(* CODESYS project Johnson,Joachim,Uppgift16.project

Project tree, tasks and I/O mapping:
  Device : CODESYS Control Win V3, 3S - Smart Software Solutions GmbH, order no. 305021, version 3.5.10.40
    application Application
      libraries: Standard, * (System)
      task MainTask (cyclic, interval t#20ms, priority 1) calls PLC_PRG
      program PLC_PRG [SFC]: MoveConv1to2, MoveCon2to3
      global variables GVL
      Symbols
*)

// Device/Application/GVL
{attribute 'qualified_only'}
VAR_GLOBAL
	// signals
	iSUB01_B1: BOOL; // Signals för conveyor 1. ontop
	iSUB02_B1: BOOL; // Signals för conveyor 2. ontop
	iSUB03_B1: BOOL; // Signals för conveyor 3. ontop
	
	// conveyor signal ontop conveyro.
	oSUB01_K1: BOOL; // MOTOR FÖR converoyr 1
	oSUB02_K1: BOOL; // MOTOR FÖR converoyr 2
	oSUB03_K1: BOOL; // MOTOR FÖR converoyr 3
END_VAR

// Device/Application/PLC_PRG
PROGRAM PLC_PRG
VAR
END_VAR
VAR // added by the converter: edge detectors and wires of the graphical bodies
    _w1, _w3 : BOOL;
    _w2 : ANY;
END_VAR

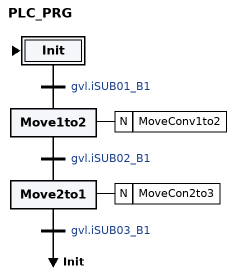
INITIAL_STEP Init:
END_STEP
TRANSITION FROM Init TO Move1to2
    := gvl.iSUB01_B1;
END_TRANSITION
STEP Move1to2:
    MoveConv1to2(N);
END_STEP
TRANSITION FROM Move1to2 TO Move2to1
    := gvl.iSUB02_B1;
END_TRANSITION
STEP Move2to1:
    MoveCon2to3(N);
END_STEP
TRANSITION FROM Move2to1 TO Init
    := gvl.iSUB03_B1;
END_TRANSITION

ACTION MoveConv1to2:
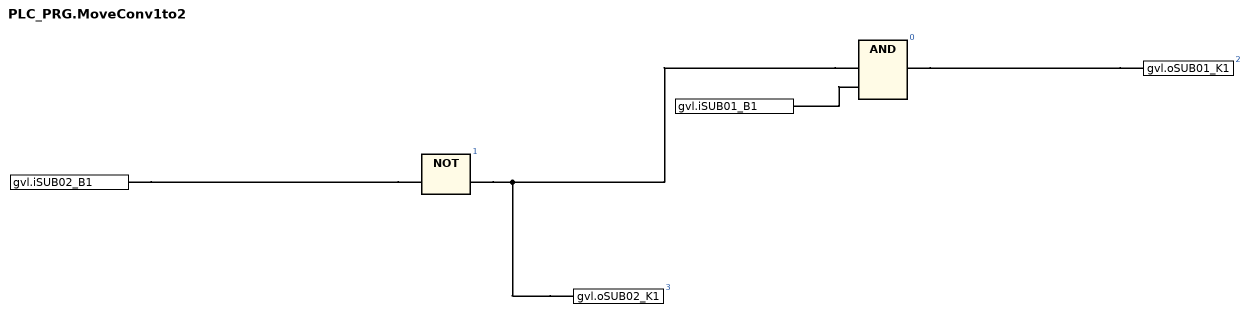
_w2 := _w1 AND gvl.iSUB01_B1;
_w1 := NOT gvl.iSUB02_B1;
gvl.oSUB01_K1 := _w2;
gvl.oSUB02_K1 := _w1;
END_ACTION

ACTION MoveCon2to3:
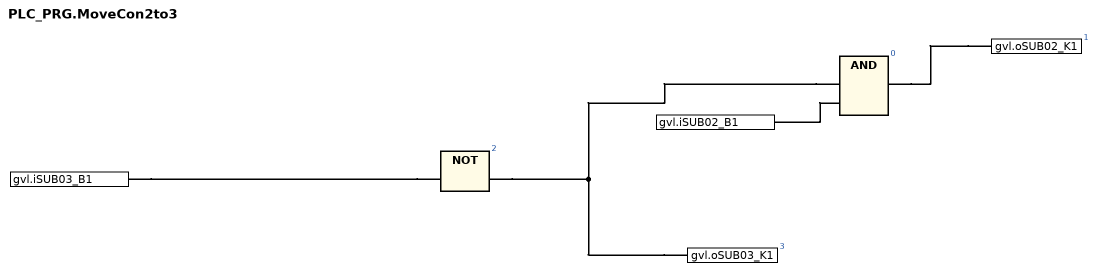
gvl.oSUB02_K1 := _w3 AND gvl.iSUB02_B1;
_w3 := NOT gvl.iSUB03_B1;
gvl.oSUB03_K1 := _w3;
END_ACTION

END_PROGRAM
